{attribute addProperty BoxType "EL2212-0000-0020"}
{attribute addProperty Id "OutputBIT10.1252TristateBIT10.1253PWMBIT10.1254ResetBIT10.1258"}
{attribute addProperty CRC "1754996918"}
{attribute addProperty SizeInBites "16"}
{attribute addProperty SizeInBytes "2"}
TYPE Control_689B20B6 :
STRUCT
	{attribute 'hide'}
	reserve_1 : BIT;
	{attribute addProperty Name "Output"}
	Output : BIT;
	{attribute addProperty Name "Tristate"}
	Tristate : BIT;
	{attribute addProperty Name "PWM"}
	PWM : BIT;
	{attribute 'hide'}
	reserve_2_BIT_0 : BIT;
	{attribute 'hide'}
	reserve_2_BIT_1 : BIT;
	{attribute 'hide'}
	reserve_2_BIT_2 : BIT;
	{attribute addProperty Name "Reset"}
	Reset : BIT;
	{attribute 'hide'}
	reserve_3 : BYTE;
END_STRUCT
END_TYPE

(* stored: Version 1.2.0.0, ProductVersion 3.1.4024.9
   DUT Control_689B20B6: Id {8c59edb1-8eb6-4c0f-8abf-1966507e9cfd} *)
